# EPICS autosave request: iocs/mythenIOC/iocBoot/iocMythen/auto_settings.req
file "ADBase_settings.req",         P=$(P),  R=cam1:
$(P)cam1:AcquireTime.PREC
file "NDFile_settings.req",         P=$(P),  R=cam1:
file "mythenV3_settings.req",       P=$(P),  R=cam1:
file "NDPluginBase_settings.req",   P=$(P),  R=image1:
file "NDStdArrays_settings.req",    P=$(P),  R=image1:
file "commonPlugin_settings.req",   P=$(P)
